(* CODESYS project Untitled1.project

Project tree, tasks and I/O mapping:
  Device : CODESYS Control Win V3, 3S - Smart Software Solutions GmbH, order no. 305021, version 3.5.11.30
    application Application
      libraries: Standard, * (System)
      task MainTask (cyclic, interval t#20ms, priority 1) calls PLC_PRG
      program PLC_PRG [FBD]
*)

// Device/Application/PLC_PRG
PROGRAM PLC_PRG
VAR
	KM: BOOL;
	TOF_0: TOF;
	S1: BOOL;
END_VAR

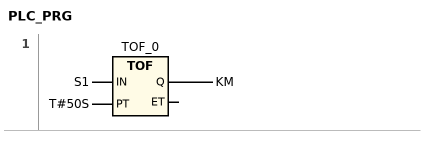
// NETWORK 1
TOF_0(IN := S1, PT := T#50S); // TOF
KM := TOF_0.Q;

END_PROGRAM
